// TwinCAT 3 PLC project SendingMQTT
// ProgramVersion: 3.1.4022.3
// libraries:
//   Tc2_Standard, * (Beckhoff Automation GmbH)
//   Tc2_System, * (Beckhoff Automation GmbH)
//   Tc2_Utilities, * (Beckhoff Automation GmbH)
//   Tc3_IotBase, * (Beckhoff Automation GmbH)
//   Tc3_IotCommunicator, * (Beckhoff Automation GmbH)
//   Tc3_JsonXml, * (Beckhoff Automation GmbH)
//   Tc3_Module, * (Beckhoff Automation GmbH)
// project tree:
//   DUTs/ TemperatureStructure.TcDUT
//   / PlcTask.TcTTO
//   POUs/ MAIN.TcPOU
// real-time tasks:
//   TASK PlcTask: cycle T#10ms, priority 20, ADS port 350
// I/O:
//   DEVICE Device 2 (EtherCAT), AmsNetId 192.168.250.2.3.1
//     Term 1 (EK1100) [EK1100 EtherCAT Coupler (2A E-Bus)]
//       Term 2 (EL1008) [EL1008 8Ch. Dig. Input 24V, 3ms]
//       Term 3 (EL2008) [EL2008 8Ch. Dig. Output 24V, 0.5A]
//       Term 4 (EL3314) [EL3314 4Ch. Ana. Input Thermocouple (TC)]
//       Term 5 (EL9011) [EL9011 End Terminal]
// variable links:
//   SendingMQTT/SendingMQTT Instance <-> Device 2 (EtherCAT)/Term 1 (EK1100)/Term 4 (EL3314)
//     PlcTask Inputs/MAIN.ai_RoomTemperature <-> TC Inputs Channel 1/Value

CONFIGURATION SendingMQTT
    RESOURCE PLC ON TwinCAT3
        TASK PlcTask(INTERVAL := T#10ms, PRIORITY := 20);
        PROGRAM MAIN WITH PlcTask : MAIN;
    END_RESOURCE
END_CONFIGURATION

// ---- DUTs/TemperatureStructure.TcDUT
TYPE TemperatureStructure :
STRUCT
	RoomTemperature : REAL;
	BathRoomTemperature : REAL;
	SomeOtherData : DINT;
END_STRUCT
END_TYPE

// ---- POUs/MAIN.TcPOU
PROGRAM MAIN
VAR
	fbMqttClient: FB_IotMqttClient; // MQTT client.       
    TopicToPublish   : STRING(255) := 'Temperatures'; // Mqtt topic on which we will broadcast the acual temperatures
    MessageToPublish : STRING(255); //String to send.
    fbSendMessageIntervalTimer : TON := (PT:=T#1S);	//Interval timer for broadcasting.
	ai_RoomTemperature AT %I* : INT; //Actual room temperature, linked to thermocouple	 
	
	TopicToPublishJson   : STRING(255) := 'Temperatures_JSON'; // Mqtt topic on which we will broadcast the acual temperatures in JSON format
	MessageToPublishJson : STRING(255); //String to send in JSON format
	fbJsonWriter : FB_JsonSaxWriter;
	fbJsonDataType : FB_JsonReadWriteDataType;
	TemperatureStructure:TemperatureStructure; 	
	  
END_VAR

IF _TaskInfo[GETCURTASKINDEXEX()].FirstCycle THEN    
    fbMqttClient.sHostName      := '192.168.178.19';
    fbMqttClient.nHostPort      := 1883;
    fbMqttClient.sTopicPrefix   := '';     
	fbMqttClient.sClientId 		:= 'Publishing PLC';
END_IF

fbMqttClient.Execute(TRUE);

IF fbMqttClient.bConnected THEN
    fbSendMessageIntervalTimer(IN:=TRUE);
    IF fbSendMessageIntervalTimer.Q THEN
        fbSendMessageIntervalTimer(IN:=FALSE);        
        MessageToPublish := CONCAT('Room temperature: ',REAL_TO_STRING(ai_RoomTemperature / 10.0));
		
        fbMqttClient.Publish(sTopic:= TopicToPublish, 
        	pPayload:= ADR(MessageToPublish), 
			nPayloadSize:= LEN2(ADR(MessageToPublish))+1, 
            eQoS:= TcIotMqttQos.AtMostOnceDelivery, 
			bRetain:= FALSE,
			bQueue:= FALSE);
			
			// Fill data
			TemperatureStructure.RoomTemperature := ai_RoomTemperature / 10.0;
			TemperatureStructure.BathRoomTemperature :=TemperatureStructure.RoomTemperature + 0.5; // No second temperature available, so this simulation value will do.
			TemperatureStructure.SomeOtherData := 33;// Random data.
			
			// COnvert to JSON string
			fbJsonWriter.ResetDocument();
			fbJsonDataType.AddJsonValueFromSymbol(fbJsonWriter, 'TemperatureStructure', SIZEOF(TemperatureStructure), ADR(TemperatureStructure));
			MessageToPublishJson := fbJsonWriter.GetDocument();
			
			//Publish
			fbMqttClient.Publish(sTopic:= TopicToPublishJson, 
        	pPayload:= ADR(MessageToPublishJson), 
			nPayloadSize:= LEN2(ADR(MessageToPublishJson))+1, 
            eQoS:= TcIotMqttQos.AtMostOnceDelivery, 
			bRetain:= FALSE,
			bQueue:= FALSE);
    END_IF
END_IF

END_PROGRAM
